INTERFACE I_SessionStorage

METHOD PUBLIC DisposeSessionDataById
VAR_INPUT
	SessionId : T_MAXSTRING;
	StorageId : T_MAXSTRING;
END_VAR
END_METHOD

METHOD PUBLIC TryRetrieveSessionDataById : BOOL
VAR_INPUT
	SessionId : T_MAXSTRING;
	StorageId : T_MAXSTRING;
	Destination : REFERENCE TO I_SessionData;
END_VAR
END_METHOD

METHOD PUBLIC TryStoreSessionDataById : BOOL
VAR_INPUT
	SessionId : T_MAXSTRING;
	StorageId : T_MAXSTRING;
	Source : I_SessionData;
END_VAR
END_METHOD

END_INTERFACE

(* stored: Version 1.1.0.1, ProductVersion 3.1.4026.18
   Itf I_SessionStorage: Id {681aeedc-281d-4081-8075-f09d2979153e}
   Method DisposeSessionDataById: Id {5e7b8d19-f2b4-4764-b133-9bbb535f46ca}
   Method TryRetrieveSessionDataById: Id {8990449f-7a3e-4565-8525-3a7a86933533}
   Method TryStoreSessionDataById: Id {5eab38a0-f4bd-424d-a9e1-847a19236fe8} *)
